Universal Robots PolyScope program: IAC003 ForceMove.urp

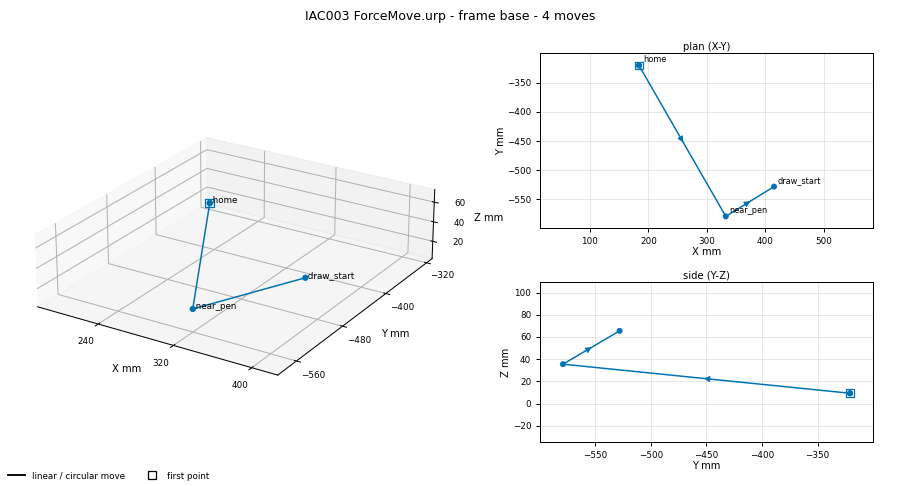
[picture p0: tool path of IAC003 ForceMove.urp in frame base, 4 of 6 moves have a stored position in this frame; points joined in program order, loops and branches not executed]
Program IAC003 ForceMove (installation=default directory=/programs createdIn=5.9.1.1031110 lastSavedIn=5.9.1.1031110 robotSerialNumber=20195501059)
Calibrated DH parameters: a=[0.000146, -0.418764, -0.053981, 0.000058, -0.000023, 0]; d=[0.162545, 37.319448, -206.067439, 168.881546, 0.09955, 0.099464]; alpha=[1.57004, -0.001979, 0.002304, 1.570607, -1.57066, 0]; deltaTheta=[0, -0.174616, -1.258233, 1.432844, -0.000001, 0]
BeforeStart
  URCap Gripper Activate (Robotiq_Grippers, Robotiq Inc.) dataModel(ResetAndActivateKey=false)
Robot Program (runOnlyOnce=true)
  URCap Gripper (Robotiq_Grippers, Robotiq Inc.) dataModel(position=69.41176470588235, force=100.0, speed=100.0, positionInDouble=69.41176470588235, forceInDouble=100.0, speedInDouble=100.0, slaveIds=[9], blocking=true)
  start_p := get_actual_tcp_pose()
  MoveJ speed 60 deg/s, acceleration 80 deg/s^2 (useActiveTCP=true) feature=Base
    Waypoint Waypoint (Variable): variable=start_p
  MoveL speed 250 mm/s, acceleration 1200 mm/s^2 (useActiveTCP=true) feature=Base
    MoveDirectionNode (selectedDirection=ZMinus) feature=Joint_6_name
      Until DISTANCE (allowActions=false deceleration=3 distanceNodeType=STOP) Distance=0.02; motionParameters(blendRadius=0)
    Waypoint home: TCP in base x=184.022 y=-320.772 z=9.398 mm, rx=0.8699 ry=3.0055 rz=-0.0545 rad; joints [98.831, -90.932, 142.715, -143.882, 269.886, 41.169] deg; TCP offset x=0 y=0 z=174 mm, rx=0 ry=0 rz=0 rad
  MoveL speed 250 mm/s, acceleration 1200 mm/s^2 (useActiveTCP=true) feature=Base
    Waypoint near_pen: TCP in base x=332.523 y=-578.911 z=35.543 mm, rx=1.6954 ry=1.6915 rz=-0.8477 rad; joints [117.47, -51.488, 119.157, -205.231, 247.172, 107.525] deg
    URCap Gripper (Robotiq_Grippers, Robotiq Inc.) dataModel(position=69.4938440492476, force=100.0, speed=100.0, positionInDouble=69.4938440492476, forceInDouble=100.0, speedInDouble=100.0, slaveIds=[9], blocking=true)
    MoveDirectionNode (selectedDirection=YMinus) feature=Base
      Until DISTANCE (allowActions=false deceleration=3 distanceNodeType=STOP) Distance=0.03; motionParameters(blendRadius=0)
    URCap Gripper (Robotiq_Grippers, Robotiq Inc.) dataModel(position=100.0, force=100.0, speed=100.0, positionInDouble=100.0, forceInDouble=100.0, speedInDouble=100.0, slaveIds=[9], blocking=true)
    MoveDirectionNode (selectedDirection=ZPlus)
      Until DISTANCE (allowActions=false deceleration=3 distanceNodeType=STOP) Distance=0.03; motionParameters(blendRadius=0)
    pen_picked := get_actual_tcp_pose()
  MoveL speed 250 mm/s, acceleration 1200 mm/s^2 (useActiveTCP=true) feature=Base
    Waypoint draw_start: TCP in base x=415.013 y=-527.991 z=65.488 mm, rx=1.6954 ry=1.6917 rz=-0.8477 rad; joints [128.702, -54.677, 115.425, -194.306, 239.14, 116.321] deg
    MoveDirectionNode (selectedDirection=ZMinus toolParams=0.01, 1.2) feature=Base
      Until TOOL_CONTACT_DETECTION (allowActions=false retraction=0 decelerationAcceleration=3 decelerationAngularAcceleration=34.906585)
    Force Frame feature=Base; selection=[0, 0, 1, 0, 0, 0]; wrench=[0, 0, -2, 0, 0, 0]; limitsForce=[0.15, 0.15, 0.15, 1.047198, 1.047198, 1.047198]; limitsMotion=[0.1, 0.1, 0.1, 0.349066, 0.349066, 0.349066]
      Wait Sleep waitTime=5
  Force Frame feature=Base; selection=[0, 0, 1, 0, 0, 0]; wrench=[0, 1, -2, 0, 0, 0]; limitsForce=[0.15, 0.15, 0.15, 1.047198, 1.047198, 1.047198]; limitsMotion=[0.1, 0.1, 0.1, 0.349066, 0.349066, 0.349066]
    MoveL speed 250 mm/s, acceleration 1200 mm/s^2 (useActiveTCP=true) feature=Base
      MoveDirectionNode (selectedDirection=XMinus toolParams=0.01, 1.2) feature=Base
        Until DISTANCE (allowActions=false deceleration=3 distanceNodeType=STOP) Distance=0.025; motionParameters(blendRadius=0)
      MoveDirectionNode (selectedDirection=YPlus toolParams=0.01, 1.2) feature=Base
        Until DISTANCE (allowActions=false deceleration=3 distanceNodeType=STOP) Distance=0.025; motionParameters(blendRadius=0)
      MoveDirectionNode (selectedDirection=XPlus toolParams=0.01, 1.2) feature=Base
        Until DISTANCE (allowActions=false deceleration=3 distanceNodeType=STOP) Distance=0.025; motionParameters(blendRadius=0)
      MoveDirectionNode (selectedDirection=YMinus toolParams=0.01, 1.2) feature=Base
        Until DISTANCE (allowActions=false deceleration=3 distanceNodeType=STOP) Distance=0.025; motionParameters(blendRadius=0)
  MoveL speed 250 mm/s, acceleration 1200 mm/s^2 (useActiveTCP=true) feature=Base
    MoveDirectionNode (selectedDirection=ZPlus) feature=Base
      Until DISTANCE (allowActions=false deceleration=3 distanceNodeType=STOP) Distance=0.025; motionParameters(blendRadius=0)
    Waypoint Waypoint (Variable): variable=pen_picked
    MoveDirectionNode (selectedDirection=ZMinus toolParams=0.01, 1.2) feature=Base
      Until TOOL_CONTACT_DETECTION (allowActions=false retraction=0 decelerationAcceleration=3 decelerationAngularAcceleration=34.906585)
    URCap Gripper (Robotiq_Grippers, Robotiq Inc.) dataModel(position=69.4938440492476, force=100.0, speed=100.0, positionInDouble=69.4938440492476, forceInDouble=100.0, speedInDouble=100.0, slaveIds=[9], blocking=true)
    MoveDirectionNode (selectedDirection=YPlus) feature=Base
      Until DISTANCE (allowActions=false deceleration=3 distanceNodeType=STOP) Distance=0.02; motionParameters(blendRadius=0)
    Waypoint home: TCP in base x=184.022 y=-320.772 z=9.398 mm, rx=0.8699 ry=3.0055 rz=-0.0545 rad; joints [98.831, -90.932, 142.715, -143.882, 269.886, 41.169] deg
